// TIA Portal V16 export
// export: Created 2023-03-29T11:04:26.9469759Z, ExportSetting WithDefaults, DisplayName Totally Integrated Automation Portal, DisplayVersion V16 Update 6, DisplayName TIA Portal Version Control Interface, DisplayVersion V16 Update 2, DisplayName TIA Portal Openness, DisplayVersion V16 Update 6, DisplayName STEP 7 Professional, DisplayVersion V16 Update 6, DisplayName STEP 7 Safety, DisplayVersion V16, DisplayName WinCC Advanced, DisplayVersion V16 Update 6
ORGANIZATION_BLOCK "Cyclic interrupt_SlaveModbusRTU"   // OB31, LAD, CyclicInterrupt
TITLE = Slave Modbus RTU
{ S7_Optimized_Access := 'TRUE' }
AUTHOR : rtecmer
VERSION : 0.1
// stored: AutoNumber true, IsIECCheckEnabled false, SetENOAutomatically false
   VAR_INPUT
      Initial_Call : Bool;   // Initial call of this OB
      Event_Count : Int;   // Events discarded
   END_VAR
BEGIN

REGION Network 1: ustawienie adresu slave PLC
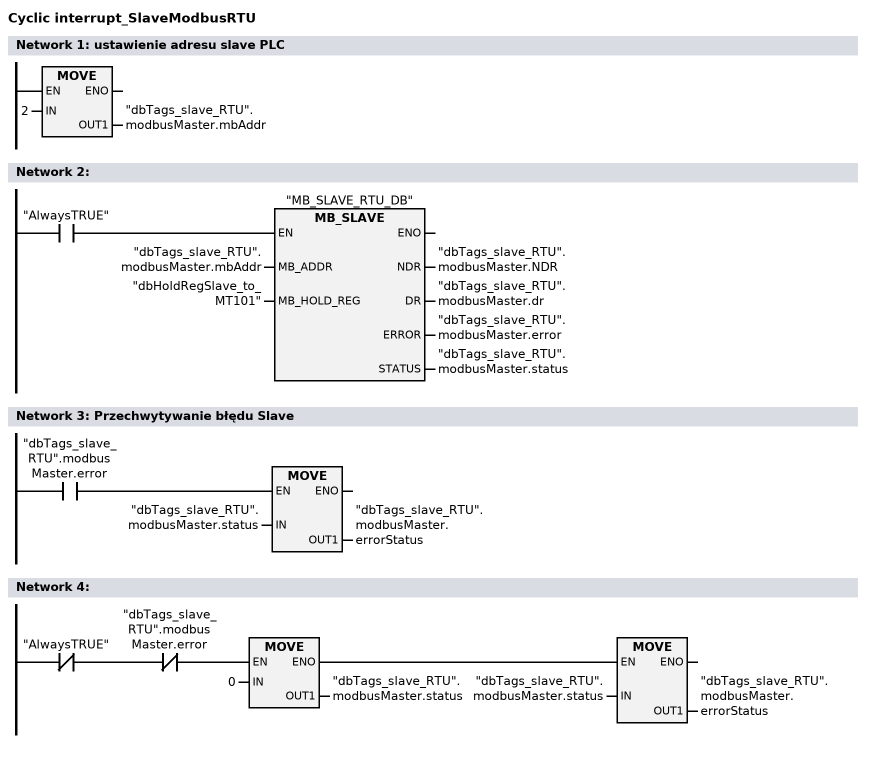
   RUNG wire#powerrail
      Move(in := 2, out1 => "dbTags_slave_RTU".modbusMaster.mbAddr)
   END_RUNG
   // the same network as SCL:
   "dbTags_slave_RTU".modbusMaster.mbAddr := 2;
END_REGION

REGION Network 2
   RUNG wire#powerrail
      Contact( "AlwaysTRUE" )
      "MB_SLAVE_RTU_DB".MB_SLAVE(MB_ADDR := "dbTags_slave_RTU".modbusMaster.mbAddr, MB_HOLD_REG := "dbHoldRegSlave_to_MT101", NDR => "dbTags_slave_RTU".modbusMaster.NDR, DR => "dbTags_slave_RTU".modbusMaster.dr, ERROR => "dbTags_slave_RTU".modbusMaster.error, STATUS => "dbTags_slave_RTU".modbusMaster.status)
   END_RUNG
   // the same network as SCL:
   IF "AlwaysTRUE" THEN
       "MB_SLAVE_RTU_DB"(MB_ADDR := "dbTags_slave_RTU".modbusMaster.mbAddr,   // MB_SLAVE
                         MB_HOLD_REG := "dbHoldRegSlave_to_MT101",
                         NDR => "dbTags_slave_RTU".modbusMaster.NDR,
                         DR => "dbTags_slave_RTU".modbusMaster.dr,
                         ERROR => "dbTags_slave_RTU".modbusMaster.error,
                         STATUS => "dbTags_slave_RTU".modbusMaster.status);
   END_IF;
END_REGION

REGION Network 3: Przechwytywanie błędu Slave
   RUNG wire#powerrail
      Contact( "dbTags_slave_RTU".modbusMaster.error )
      Move(in := "dbTags_slave_RTU".modbusMaster.status, out1 => "dbTags_slave_RTU".modbusMaster.errorStatus)
   END_RUNG
   // the same network as SCL:
   IF "dbTags_slave_RTU".modbusMaster.error THEN
       "dbTags_slave_RTU".modbusMaster.errorStatus := "dbTags_slave_RTU".modbusMaster.status;
   END_IF;
END_REGION

REGION Network 4
   RUNG wire#powerrail
      I_Contact( "AlwaysTRUE" )
      I_Contact( "dbTags_slave_RTU".modbusMaster.error )
      Move(in := 0, out1 => "dbTags_slave_RTU".modbusMaster.status)
      Move(in := "dbTags_slave_RTU".modbusMaster.status, out1 => "dbTags_slave_RTU".modbusMaster.errorStatus)
   END_RUNG
   // the same network as SCL:
   IF NOT "AlwaysTRUE" AND NOT "dbTags_slave_RTU".modbusMaster.error THEN
       "dbTags_slave_RTU".modbusMaster.status := 0;
       "dbTags_slave_RTU".modbusMaster.errorStatus := "dbTags_slave_RTU".modbusMaster.status;
   END_IF;
END_REGION
END_ORGANIZATION_BLOCK
